FUNCTION_BLOCK bfb_sat_classifier
  (* Standard: 61499-2 *)
  (* Version 0.1, 2018-00-07, hpea485, UOA *)
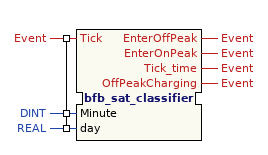
  EVENT_INPUT
    Tick WITH Minute, day;
  END_EVENT
  EVENT_OUTPUT
    EnterOffPeak;
    EnterOnPeak;
    Tick_time;
    OffPeakCharging;
  END_EVENT
  VAR_INPUT
    Minute : DINT;
    day : REAL;
  END_VAR
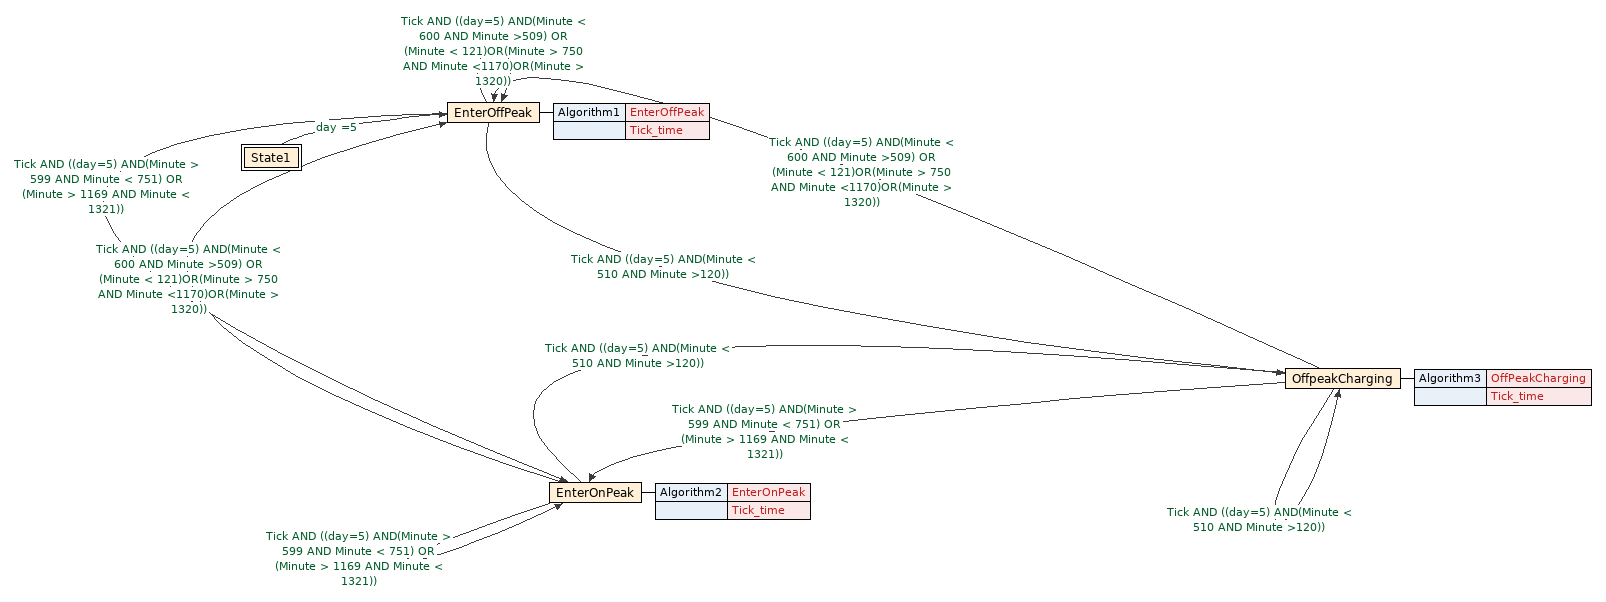
  EC_STATES
    State1;
    EnterOffPeak : Algorithm1 -> EnterOffPeak, -> Tick_time;
    EnterOnPeak : Algorithm2 -> EnterOnPeak, -> Tick_time;
    OffpeakCharging : Algorithm3 -> OffPeakCharging, -> Tick_time;
  END_STATES
  EC_TRANSITIONS
    EnterOffPeak TO EnterOffPeak := Tick AND ((day=5) AND(Minute < 600 AND Minute >509) OR (Minute < 121)OR(Minute > 750 AND Minute <1170)OR(Minute > 1320));
    EnterOffPeak TO EnterOnPeak := Tick AND ((day=5) AND(Minute > 599 AND Minute < 751) OR (Minute > 1169  AND Minute < 1321));
    EnterOffPeak TO OffpeakCharging := Tick AND ((day=5) AND(Minute < 510 AND Minute >120));
    EnterOnPeak TO EnterOffPeak := Tick AND ((day=5) AND(Minute < 600 AND Minute >509) OR (Minute < 121)OR(Minute > 750 AND Minute <1170)OR(Minute > 1320));
    EnterOnPeak TO EnterOnPeak := Tick AND ((day=5) AND(Minute > 599 AND Minute < 751) OR (Minute > 1169  AND Minute < 1321));
    EnterOnPeak TO OffpeakCharging := Tick AND ((day=5) AND(Minute < 510 AND Minute >120));
    OffpeakCharging TO EnterOnPeak := Tick AND ((day=5) AND(Minute > 599 AND Minute < 751) OR (Minute > 1169  AND Minute < 1321));
    OffpeakCharging TO OffpeakCharging := Tick AND ((day=5) AND(Minute < 510 AND Minute >120));
    OffpeakCharging TO EnterOffPeak := Tick AND ((day=5) AND(Minute < 600 AND Minute >509) OR (Minute < 121)OR(Minute > 750 AND Minute <1170)OR(Minute > 1320));
    State1 TO EnterOffPeak := day =5;
  END_TRANSITIONS
  ALGORITHM Algorithm1 IN C:
printf("Entered OFF PEAK.....\r\n");
  END_ALGORITHM
  ALGORITHM Algorithm2 IN C:
printf(" Entered On peak .....\r\n ");
  END_ALGORITHM
  ALGORITHM Algorithm3 IN C:
printf(" OffPeak Charging \r\n ");
  END_ALGORITHM
END_FUNCTION_BLOCK
